Universal Robots PolyScope program: RG2_SubP.urp

ProgramRoot setBeforeStartSequence=true; directory=/programs; name=RG2_SubP; programVersion=(project__name=PolyScope, major__version=1, minor__version=5, svn__revision=7727, build__date=Jan 23 2012, 10:38:07); robotEnvironmentFileName=default
  BeforeStart description=<html>This sequence will execute before the main program.</html>; name=BeforeStart
    Popup type=MESSAGE
    Halt 
  MainProgram cartesianAcceleration=0.0; cartesianSpeed=0.0; jointAcceleration=0.0; jointSpeed=0.0; moveAsFastAsPossible=true; sharedProcessMoveBlendRadius=0.025; featureReference=(installationNameReference=Base); motionType=JOINT_SPACE
    Assignment assignmentValueSource=0; assignmentOperatorMessage=110; expr=110; operatorValueType=INTEGER; valueSource=EXPRESSION; variable=(name=Open, prefersPersistentValue=false, requestANewUniqueName=false)
    Assignment assignmentValueSource=0; assignmentOperatorMessage=10; expr=10; operatorValueType=INTEGER; valueSource=EXPRESSION; variable=(name=Close, prefersPersistentValue=false, requestANewUniqueName=false)
    Folder name=RG2 settings
      Assignment assignmentValueSource=0; assignmentOperatorMessage=40; expr=40; operatorValueType=INTEGER; valueSource=EXPRESSION; variable=(name=Force_, prefersPersistentValue=false, requestANewUniqueName=false)
      Assignment assignmentValueSource=0; assignmentOperatorMessage=60; expr=60; operatorValueType=INTEGER; valueSource=EXPRESSION; variable=(name=Open2, prefersPersistentValue=false, requestANewUniqueName=false)
      Assignment assignmentValueSource=0; assignmentOperatorMessage=50; expr=50; operatorValueType=INTEGER; valueSource=EXPRESSION; variable=(name=Close2, prefersPersistentValue=false, requestANewUniqueName=false)
      Assignment assignmentValueSource=0; assignmentOperatorMessage=40; expr=40; operatorValueType=INTEGER; valueSource=EXPRESSION; variable=(name=Force2, prefersPersistentValue=false, requestANewUniqueName=false)
    Script type=1; scriptFile=/programs/program_RG2.script
    Script type=1; scriptFile=/programs/open.script
